FUNCTION UpdateEventTimeStamp : ST_Event
VAR_INPUT
	stEvent : REFERENCE TO ST_Event ;
END_VAR

VAR
	fbgetsystemtime: GETSYSTEMTIME;
	stFileTime : T_FILETIME;
	nHigh : UDINT;
	nLow : UDINT;	
END_VAR

fbgetsystemtime(timeLodw=>stFileTime.dwLowDateTime , timeHidw=>stFileTime.dwHighDateTime); 

stEvent.dtTimestamp:=FILETIME_TO_DT(stFileTime);

END_FUNCTION

(* stored: Version 1.1.0.1, ProductVersion 3.1.4024.12
   POU UpdateEventTimeStamp: Id {bfbf6de3-9080-4c3c-aa80-ea670f53c0a7}, SpecialFunc None *)
